TYPE CylinderStatus :
STRUCT
	ActionDescription : STRING(100);	
END_STRUCT
END_TYPE

(* stored: Version 1.1.0.1
   DUT CylinderStatus: Id {c1c6431e-77ff-0e62-0580-b5148e9ff6d7} *)
